FUNCTION_BLOCK ReadJSON (* Decode JSON string *)
  (* Standard: 61499-2; Description: Copyright (c) 2026 Thomas Mayr This program and the accompanying materials are made available under the terms of the Eclipse Public License 2.0 which is available at https://www.eclipse.org/legal/epl-2.0/ SPDX-License-Identifier: EPL-2.0 *)
  (* Version 1.0, 2026-05-16, Thomas Mayr *)
  PACKAGE eclipse4diac::convert;
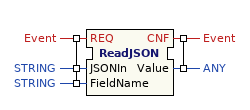
  EVENT_INPUT
    REQ WITH JSONIn, FieldName; (* Execute *)
  END_EVENT
  EVENT_OUTPUT
    CNF WITH Value; (* Execution done *)
  END_EVENT
  VAR_INPUT
    JSONIn : STRING; (* Input JSON string *)
    FieldName : STRING; (* Field to extract *)
  END_VAR
  VAR_OUTPUT
    Value : ANY; (* Extracted field value *)
  END_VAR
END_FUNCTION_BLOCK
